FUNCTION_BLOCK PUBLIC EcMasterFrameStats IMPLEMENTS IEcTask
VAR_INPUT
END_VAR
VAR_OUTPUT
END_VAR
VAR
	iState : INT;
	masterFrameStats : Tc2_EtherCAT.FB_EcMasterFrameStatistic;
	_execute: BOOL;
	_done: BOOL;
	_busy: BOOL;
	_error: BOOL;
	_netId: AMSNETID;
END_VAR

CASE iState OF
	0:
		IF _execute THEN
			_done := FALSE;
			_busy := TRUE;
			_error := FALSE;
			masterFrameStats.bExecute := TRUE;
			IF masterFrameStats.bBusy THEN
				iState := 10;
				_execute := false;
			END_IF
		END_IF
	10:
		IF NOT masterFrameStats.bBusy THEN
			IF NOT masterFrameStats.bError THEN
				_done := TRUE;
			ELSE
				_error := TRUE;
			END_IF
			_busy := FALSE;
			masterFrameStats.bExecute := FALSE;
			iState := 0;
		END_IF
END_CASE

masterFrameStats(sNetId := Tc2_System.F_CreateAmsNetId(nIds := NetId));

{warning 'add method implementation '}
METHOD Abort : BOOL
masterFrameStats.bExecute := FALSE;
_busy := FALSE;
_execute := FALSE;
Abort := TRUE;
iState := 0;
END_METHOD

{warning 'add property implementation'}
PROPERTY Busy : BOOL
GET
Busy := _busy;
END_GET
END_PROPERTY

{warning 'add property implementation'}
PROPERTY Done : BOOL
GET
Done := _done;
END_GET
END_PROPERTY

{warning 'add property implementation'}
PROPERTY Error : BOOL
GET
Error := _error;
END_GET
END_PROPERTY

METHOD Execute : BOOL
VAR_INPUT
END_VAR
IF NOT Busy THEN
	Execute := _execute := TRUE;
END_IF
END_METHOD

PROPERTY FramesPerSecond  : LREAL
GET
FramesPerSecond := masterFrameStats.fFramesPerSecond;
END_GET
END_PROPERTY

PROPERTY LostFrames : UDINT
GET
LostFrames := masterFrameStats.nLostFrames;
END_GET
END_PROPERTY

PROPERTY LostQueuedFrames : udint
GET
LostQueuedFrames := masterFrameStats.nLostQueuedFrames;
END_GET
END_PROPERTY

{warning 'add property implementation'}
PROPERTY NetID : amsnetid
GET
NetID := _netId;
END_GET
SET
_netId := NetID;
END_SET
END_PROPERTY

PROPERTY QueuedFramesPerSecond : lreal
GET
QueuedFramesPerSecond := masterFrameStats.fQueuedFramesPerSecond;
END_GET
END_PROPERTY

END_FUNCTION_BLOCK

(* stored: Version 1.1.0.1, ProductVersion 3.1.4024.9
   POU EcMasterFrameStats: Id {4f2a2d5c-80f9-4ad1-9f7a-af400c885aba}, SpecialFunc None
   Method Abort: Id {24b69794-6527-4c60-a685-0294a95d95f0}
   Property Busy: Id {92baef78-27be-417d-a5e4-b7e3718f9c68}
   Get Get: Id {4b22d7e6-5242-4388-9ce3-10ba30296c80}
   Property Done: Id {b10ec56c-2400-442f-bd76-9433de1cc8c7}
   Get Get: Id {ccbf4283-da75-4218-b4df-f93ea812e672}
   Property Error: Id {4c59c668-a8c2-4bcd-b913-b9e64d8dabfd}
   Get Get: Id {00bfd487-54b8-4e10-8cc7-00ae0db37bf7}
   Method Execute: Id {1ee721c9-aafc-4c87-8ca9-32345a53bd3b}
   Property FramesPerSecond: Id {916a482e-24f7-4585-af91-5ce29a0c546d}
   Get Get: Id {ed96813f-77ca-468b-9b04-2d5f570e54e3}
   Property LostFrames: Id {667e091e-12ee-49bc-8f27-11506f0442c4}
   Get Get: Id {07ded8b8-172f-4f43-991b-94ed349d3f77}
   Property LostQueuedFrames: Id {1b626e3f-3519-47ba-b2d6-0076a80e8d7d}
   Get Get: Id {d6217ef2-16ea-481f-abc7-ca2e6a34da18}
   Property NetID: Id {b62dd98e-416b-4db7-83b6-89191f515461}
   Get Get: Id {d9d16ba9-78c5-4f4c-b1c4-ab6fbe3aadc0}
   Set Set: Id {74e2852f-7467-44b1-8dc2-9441abb0f8c2}
   Property QueuedFramesPerSecond: Id {3cc27eed-9c7a-4344-bab3-ce383ede3dee}
   Get Get: Id {9ab89b5e-7df3-42c3-8392-072a465db611} *)
